INTERFACE I_UniversalAxis

PROPERTY Active : REFERENCE TO BOOL
GET
END_GET
END_PROPERTY

PROPERTY Error : REFERENCE TO BOOL
GET
END_GET
END_PROPERTY

(* Copy it to derived Function block if developing this function *)
PROPERTY ErrorID : REFERENCE TO UDINT
GET
END_GET
END_PROPERTY

METHOD MR_Abort : BOOL
END_METHOD

METHOD MR_Init : BOOL
END_METHOD

METHOD MR_Reset : BOOL
END_METHOD

(* Copy it to derived Function block if developing this function *)
PROPERTY Name : STRING
GET
END_GET
SET
END_SET
END_PROPERTY

{attribute 'to_string'}
PROPERTY State : REFERENCE TO E_AxisState
GET
END_GET
END_PROPERTY

END_INTERFACE

(* stored: Version 1.1.0.1, ProductVersion 3.1.4024.12
   Itf I_UniversalAxis: Id {8e427913-59b3-4d06-887a-4072fb08d6c0}
   Property Active: Id {a649d022-91f1-412a-8e03-b31ea5ba4b97}
   Get Get: Id {a4122a89-64ba-40bf-8b93-a6150501d41a}
   Property Error: Id {5fd1ffb0-7593-4fff-a0ad-e35dfc2e2777}
   Get Get: Id {5951bb7b-f3b2-4424-aebb-b6a84236b8f1}
   Property ErrorID: Id {70152098-3716-413a-8ea0-a71ad208d89f}
   Get Get: Id {3b2e3ccf-619d-40f7-9f5b-b74efc8c41cb}
   Method MR_Abort: Id {2d6f31f7-b221-40f9-a6fa-79a04dce778a}
   Method MR_Init: Id {b7d863a9-e9f4-4383-bab7-e39162e0c718}
   Method MR_Reset: Id {fd624c9b-c86b-4c51-ada4-da9d67891b35}
   Property Name: Id {46be5bf4-905e-4f1e-b29e-b8f780078568}
   Get Get: Id {a23bcdfa-a40e-45a0-bd97-329ecdda126e}
   Set Set: Id {826a4881-a8e4-4867-989f-fd1cdd911533}
   Property State: Id {91b2d6bb-3a85-4a51-a619-90fec7684f0d}
   Get Get: Id {a8157ad4-c10a-474d-9072-eb29727172e0} *)
